FUNCTION didSensorChange : BOOL
VAR_INPUT
	readTemp			: 	readTemp2;
	whichSwitch			:	switch2;
END_VAR
VAR
END_VAR

IF readTemp.fbRecGeneric.bReceive = FALSE OR whichSwitch.fbRecGeneric.bReceive = FALSE THEN
	didSensorChange := TRUE;
	ELSE
		didSensorChange := FALSE;
END_IF

END_FUNCTION

(* stored: Version 1.1.0.1, ProductVersion 3.1.4024.2
   POU didSensorChange: Id {49137ea6-73fe-475b-8be3-85a537fd34d6}, SpecialFunc None *)
